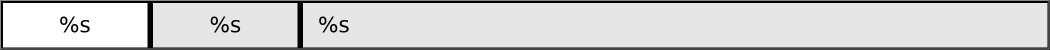
VISUALIZATION AlarmRow  // 1050x50
VAR_IN_OUT

	
END_VAR

VAR_INPUT
	sAlarmTextList 	: STRING;
	sEventDataTextList : STRING;
	stAlarmLogEvent : ST_AlarmEventData_TextList;
END_VAR
    Rectangle (0,0 150x50), "%s", text variable: stAlarmLogEvent.sTime, colour toggle: stAlarmLogEvent.iClass = 7
    Rectangle (300,0 750x50), colour toggle: stAlarmLogEvent.iClass = 7, text list: ''
    Rectangle (150,0 150x50), colour toggle: stAlarmLogEvent.iClass = 7, text list: ''
    Textfield (315,10 721x30), "%s", invisible if: stAlarmLogEvent.diEventID = 0, text list: sAlarmTextList, text index: stAlarmLogEvent.diEventID
    Textfield (159,10 133x30), "%s", invisible if: stAlarmLogEvent.diEventID = 0, text list: sEventDataTextList, text index: stAlarmLogEvent.iClass
END_VISUALIZATION

(* stored: Version 1.1.0.1
   Visu AlarmRow: Id {802d672e-5c7b-44cd-a141-cb4fad3ea135} *)
